TYPE ST_CAMERA_ImageData :
STRUCT
	nCodesRead		: INT;
	tScanTime		: TIME;		(* image cycle time (including image acquisition time and decode time) *)
	sDecodeStatus	: T_MaxString;
	stTriggerID		: ST_CAMERA_TriggerID;
	aCodeData		: ARRAY[1..cMAX_CAMERA_PROG_NUMBER] OF ST_CAMERA_CodeData;
END_STRUCT
END_TYPE

(* stored: Version 1.1.0.1
   DUT ST_CAMERA_ImageData: Id {744e136a-df5c-43a7-a2a4-5fbaebd6b786} *)
